// TIA Portal V21 export
FUNCTION "InvertBit" : Void   // FC901, LAD
{ S7_Optimized_Access := 'TRUE' }
// stored: AutoNumber false, SetENOAutomatically false
   VAR_IN_OUT
      Bit : Bool;
   END_VAR
BEGIN

REGION Network 1
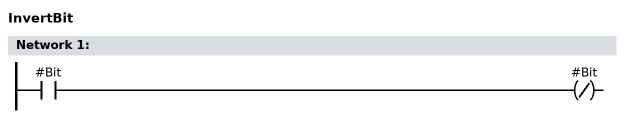
   RUNG wire#powerrail
      Contact( #Bit )
      I_Coil( #Bit )
   END_RUNG
   // the same network as SCL:
   #Bit := NOT #Bit;
END_REGION
END_FUNCTION
